LIN {X -403.787,Y 333.050,Z -17.519,A 0.015,B -0.000,C 180.000} C_DIS
LIN {X -401.252,Y 328.076,Z -17.721,A 0.015,B -0.000,C -180.000} C_DIS
LIN {X -395.738,Y 327.203,Z -17.924,A 0.015,B 0.000,C -180.000} C_DIS
LIN {X -391.790,Y 331.150,Z -18.126,A 0.015,B 0.000,C 180.000} C_DIS
LIN {X -392.664,Y 336.664,Z -18.328,A 0.015,B -0.000,C -180.000} C_DIS
LIN {X -397.638,Y 339.199,Z -18.531,A 0.015,B 0.000,C 180.000} C_DIS
LIN {X -398.507,Y 339.199,Z -18.561,A 0.015,B -0.000,C 180.000} C_DIS
LIN {X -399.336,Y 339.133,Z -18.590,A 0.015,B -0.000,C -180.000} C_DIS
LIN {X -399.692,Y 339.076,Z -18.603,A 0.015,B -0.000,C -180.000} C_DIS
LIN {X -400.552,Y 338.848,Z -18.634,A 0.015,B 0.000,C 180.000} C_DIS
LIN {X -400.596,Y 338.832,Z -18.635,A 0.015,B 0.000,C -180.000} C_DIS
LIN {X -401.281,Y 338.494,Z -18.662,A 0.015,B 0.000,C 180.000} C_DIS
LIN {X -401.404,Y 338.418,Z -18.667,A 0.015,B 0.000,C 180.000} C_DIS
LIN {X -402.842,Y 337.053,Z -18.737,A 0.015,B -0.000,C 180.000} C_DIS
LIN {X -402.866,Y 337.018,Z -18.738,A 0.015,B 0.000,C -180.000} C_DIS
LIN {X -403.753,Y 334.430,Z -18.835,A 0.015,B -0.000,C -180.000} C_DIS
LIN {X -403.779,Y 333.946,Z -18.852,A 0.015,B -0.000,C -180.000} C_DIS
LIN {X -403.787,Y 333.653,Z -18.862,A 0.015,B -0.000,C -180.000} C_DIS
LIN {X -403.787,Y 333.050,Z -18.883,A 0.015,B 0.000,C -180.000} C_DIS
LIN {X -401.252,Y 328.076,Z -19.086,A 0.015,B -0.000,C 180.000} C_DIS
LIN {X -395.738,Y 327.203,Z -19.288,A 0.015,B 0.000,C -180.000} C_DIS
LIN {X -391.790,Y 331.150,Z -19.491,A 0.015,B 0.000,C 180.000} C_DIS
LIN {X -392.664,Y 336.664,Z -19.693,A 0.015,B -0.000,C -180.000} C_DIS
LIN {X -397.638,Y 339.199,Z -19.895,A 0.015,B 0.000,C 180.000} C_DIS
LIN {X -398.507,Y 339.199,Z -19.926,A 0.015,B 0.000,C -180.000} C_DIS
LIN {X -399.336,Y 339.133,Z -19.955,A 0.015,B -0.000,C 180.000} C_DIS
LIN {X -399.692,Y 339.076,Z -19.967,A 0.015,B -0.000,C 180.000} C_DIS
LIN {X -400.552,Y 338.848,Z -19.998,A 0.015,B -0.000,C 180.000} C_DIS
LIN {X -400.596,Y 338.832,Z -20.000,A 0.015,B 0.000,C 180.000} C_DIS
LIN {X -400.134,Y 339.006,Z -20.000,A 0.015,B -0.000,C 180.000} C_DIS
LIN {X -398.924,Y 339.199,Z -20.000,A 0.015,B 0.000,C 180.000} C_DIS
LIN {X -213.196,Y 339.203,Z -20.000,A 0.015,B 0.000,C 180.000} C_DIS
LIN {X -213.589,Y 339.144,Z -20.000,A 0.015,B -0.000,C 180.000} C_DIS
LIN {X -214.096,Y 339.026,Z -20.000,A 0.015,B 0.000,C 180.000} C_DIS
LIN {X -215.185,Y 338.684,Z -20.000,A 0.015,B 0.000,C 180.000} C_DIS
LIN {X -215.676,Y 338.486,Z -20.000,A 0.015,B -0.000,C -180.000} C_DIS
LIN {X -226.923,Y 332.891,Z -20.000,A 0.015,B 0.000,C 180.000} C_DIS
LIN {X -227.590,Y 332.454,Z -20.000,A 0.015,B 0.000,C -180.000} C_DIS
LIN {X -228.678,Y 331.541,Z -20.000,A 0.015,B 0.000,C 180.000} C_DIS
LIN {X -228.854,Y 331.383,Z -20.000,A 0.015,B -0.000,C 180.000} C_DIS
LIN {X -237.260,Y 323.263,Z -20.000,A 0.015,B 0.000,C -180.000} C_DIS
LIN {X -237.740,Y 322.682,Z -20.000,A 0.015,B 0.000,C -180.000} C_DIS
LIN {X -238.689,Y 321.231,Z -20.000,A 0.015,B -0.000,C -180.000} C_DIS
LIN {X -238.828,Y 321.000,Z -20.000,A 0.015,B 0.000,C -180.000} C_DIS
LIN {X -243.976,Y 311.569,Z -20.000,A 0.015,B -0.000,C 180.000} C_DIS
LIN {X -244.137,Y 311.231,Z -20.000,A 0.015,B 0.000,C -180.000} C_DIS
LIN {X -244.732,Y 309.780,Z -20.000,A 0.015,B -0.000,C 180.000} C_DIS
LIN {X -244.946,Y 309.009,Z -20.000,A 0.015,B 0.000,C 180.000} C_DIS
LIN {X -246.389,Y 299.577,Z -20.000,A 0.015,B 0.000,C 180.000} C_DIS
LIN {X -246.415,Y 299.356,Z -20.000,A 0.015,B -0.000,C 180.000} C_DIS
LIN {X -246.509,Y 298.268,Z -20.000,A 0.015,B -0.000,C -180.000} C_DIS
CIRC {X -246.514,Y 297.749,Z -20.000,A 0.015,B 0.000,C -180.000},{X -246.439,Y 297.235,Z -20.000,A 0.015,B 0.000,C -180.000} C_DIS
LIN {X -245.041,Y 291.021,Z -20.000,A 0.015,B 0.000,C 180.000} C_DIS
LIN {X -245.028,Y 290.962,Z -20.000,A 0.015,B 0.000,C 180.000} C_DIS
LIN {X -244.067,Y 287.020,Z -20.000,A 0.015,B 0.000,C 180.000} C_DIS
LIN {X -243.752,Y 286.205,Z -20.000,A 0.015,B 0.000,C -180.000} C_DIS
LIN {X -242.372,Y 283.666,Z -20.000,A 0.015,B 0.000,C 180.000} C_DIS
LIN {X -242.162,Y 283.330,Z -20.000,A 0.015,B -0.000,C -180.000} C_DIS
LIN {X -239.169,Y 279.093,Z -20.000,A 0.015,B 0.000,C -180.000} C_DIS
LIN {X -239.003,Y 278.877,Z -20.000,A 0.015,B 0.000,C -180.000} C_DIS
LIN {X -237.090,Y 276.585,Z -20.000,A 0.015,B -0.000,C -180.000} C_DIS
LIN {X -236.752,Y 276.235,Z -20.000,A 0.015,B 0.000,C -180.000} C_DIS
LIN {X -236.388,Y 275.908,Z -20.000,A 0.015,B -0.000,C -180.000} C_DIS
LIN {X -236.084,Y 275.665,Z -20.000,A 0.015,B 0.000,C 180.000} C_DIS
LIN {X -232.452,Y 273.091,Z -20.000,A 0.015,B 0.000,C -180.000} C_DIS
LIN {X -232.331,Y 273.008,Z -20.000,A 0.015,B -0.000,C -180.000} C_DIS
LIN {X -229.064,Y 270.900,Z -20.000,A 0.015,B 0.000,C -180.000} C_DIS
LIN {X -228.750,Y 270.720,Z -20.000,A 0.015,B -0.000,C 180.000} C_DIS
LIN {X -227.172,Y 269.926,Z -20.000,A 0.015,B 0.000,C -180.000} C_DIS
LIN {X -226.775,Y 269.757,Z -20.000,A 0.015,B 0.000,C -180.000} C_DIS
LIN {X -224.725,Y 269.036,Z -20.000,A 0.015,B 0.000,C 180.000} C_DIS
LIN {X -224.251,Y 268.907,Z -20.000,A 0.015,B 0.000,C 180.000} C_DIS
LIN {X -219.172,Y 267.914,Z -20.000,A 0.015,B 0.000,C -180.000} C_DIS
LIN {X -218.973,Y 267.881,Z -20.000,A 0.015,B 0.000,C 180.000} C_DIS
LIN {X -215.345,Y 267.394,Z -20.000,A 0.015,B 0.000,C 180.000} C_DIS
LIN {X -214.895,Y 267.364,Z -20.000,A 0.015,B 0.000,C 180.000} C_DIS
LIN {X -178.617,Y 267.364,Z -20.000,A 0.015,B 0.000,C 180.000} C_DIS
LIN {X -178.167,Y 267.394,Z -20.000,A 0.015,B -0.000,C 180.000} C_DIS
LIN {X -174.539,Y 267.881,Z -20.000,A 0.015,B -0.000,C 180.000} C_DIS
LIN {X -174.340,Y 267.914,Z -20.000,A 0.015,B 0.000,C -180.000} C_DIS
LIN {X -169.261,Y 268.907,Z -20.000,A 0.015,B 0.000,C 180.000} C_DIS
LIN {X -168.860,Y 269.012,Z -20.000,A 0.015,B 0.000,C 180.000} C_DIS
LIN {X -167.472,Y 269.465,Z -20.000,A 0.015,B 0.000,C -180.000} C_DIS
LIN {X -167.129,Y 269.598,Z -20.000,A 0.015,B 0.000,C -180.000} C_DIS
LIN {X -165.283,Y 270.432,Z -20.000,A 0.015,B 0.000,C -180.000} C_DIS
LIN {X -164.859,Y 270.662,Z -20.000,A 0.015,B 0.000,C -180.000} C_DIS
LIN {X -161.562,Y 272.763,Z -20.000,A 0.015,B 0.000,C -180.000} C_DIS
LIN {X -161.461,Y 272.830,Z -20.000,A 0.015,B 0.000,C -180.000} C_DIS
LIN {X -158.559,Y 274.828,Z -20.000,A 0.015,B 0.000,C 180.000} C_DIS
LIN {X -158.397,Y 274.947,Z -20.000,A 0.015,B 0.000,C -180.000} C_DIS
LIN {X -156.938,Y 276.085,Z -20.000,A 0.015,B 0.000,C -180.000} C_DIS
LIN {X -156.452,Y 276.549,Z -20.000,A 0.015,B 0.000,C -180.000} C_DIS
LIN {X -155.008,Y 278.233,Z -20.000,A 0.015,B -0.000,C 180.000} C_DIS
LIN {X -154.823,Y 278.469,Z -20.000,A 0.015,B -0.000,C 180.000} C_DIS
LIN {X -151.360,Y 283.315,Z -20.000,A 0.015,B -0.000,C 180.000} C_DIS
LIN {X -151.140,Y 283.666,Z -20.000,A 0.015,B 0.000,C 180.000} C_DIS
LIN {X -149.760,Y 286.205,Z -20.000,A 0.015,B -0.000,C 180.000} C_DIS
LIN {X -149.440,Y 287.040,Z -20.000,A 0.015,B 0.000,C -180.000} C_DIS
LIN {X -147.117,Y 296.834,Z -20.000,A 0.015,B 0.000,C -180.000} C_DIS
LIN {X -147.030,Y 297.450,Z -20.000,A 0.015,B -0.000,C 180.000} C_DIS
LIN {X -146.995,Y 298.175,Z -20.000,A 0.015,B 0.000,C 180.000} C_DIS
LIN {X -147.027,Y 298.837,Z -20.000,A 0.015,B 0.000,C 180.000} C_DIS
LIN {X -148.481,Y 308.631,Z -20.000,A 0.015,B 0.000,C 180.000} C_DIS
LIN {X -148.624,Y 309.222,Z -20.000,A 0.015,B 0.000,C 180.000} C_DIS
LIN {X -149.116,Y 310.673,Z -20.000,A 0.015,B 0.000,C 180.000} C_DIS
LIN {X -149.349,Y 311.203,Z -20.000,A 0.015,B -0.000,C -180.000} C_DIS
LIN {X -154.682,Y 320.997,Z -20.000,A 0.015,B 0.000,C -180.000} C_DIS
LIN {X -154.822,Y 321.231,Z -20.000,A 0.015,B 0.000,C -180.000} C_DIS
LIN {X -155.772,Y 322.682,Z -20.000,A 0.015,B 0.000,C 180.000} C_DIS
LIN {X -156.247,Y 323.258,Z -20.000,A 0.015,B 0.000,C 180.000} C_DIS
LIN {X -163.722,Y 330.512,Z -20.000,A 0.015,B 0.000,C 180.000} C_DIS
LIN {X -163.842,Y 330.624,Z -20.000,A 0.015,B 0.000,C 180.000} C_DIS
LIN {X -165.860,Y 332.401,Z -20.000,A 0.015,B 0.000,C -180.000} C_DIS
LIN {X -166.589,Y 332.891,Z -20.000,A 0.015,B -0.000,C 180.000} C_DIS
LIN {X -177.836,Y 338.486,Z -20.000,A 0.015,B 0.000,C 180.000} C_DIS
LIN {X -178.194,Y 338.639,Z -20.000,A 0.015,B 0.000,C -180.000} C_DIS
LIN {X -178.919,Y 338.901,Z -20.000,A 0.015,B 0.000,C -180.000} C_DIS
LIN {X -179.549,Y 339.062,Z -20.000,A 0.015,B 0.000,C 180.000} C_DIS
LIN {X -180.468,Y 339.204,Z -20.000,A 0.015,B 0.000,C -180.000} C_DIS
LIN {X 4.865,Y 339.209,Z -20.000,A 0.015,B -0.000,C -180.000} C_DIS
LIN {X 5.937,Y 339.152,Z -20.000,A 0.015,B -0.000,C 180.000} C_DIS
LIN {X 6.802,Y 338.955,Z -20.000,A 0.015,B 0.000,C 180.000} C_DIS
LIN {X 7.069,Y 338.840,Z -20.000,A 0.015,B 0.000,C 180.000} C_DIS
LIN {X 7.374,Y 338.634,Z -20.000,A 0.015,B -0.000,C 180.000} C_DIS
LIN {X 9.664,Y 336.377,Z -20.000,A 0.015,B 0.000,C -180.000} C_DIS
LIN {X 9.898,Y 336.018,Z -20.000,A 0.015,B 0.000,C -180.000} C_DIS
LIN {X 10.072,Y 335.556,Z -20.000,A 0.015,B -0.000,C -180.000} C_DIS
LIN {X 10.265,Y 334.347,Z -20.000,A 0.015,B -0.000,C 180.000} C_DIS
LIN {X 10.273,Y 31.658,Z -20.000,A 0.015,B 0.000,C -180.000} C_DIS
LIN {X 8.905,Y 37.176,Z -20.000,A 0.015,B 0.000,C 180.000} C_DIS
LIN {X 8.665,Y 37.838,Z -20.000,A 0.015,B 0.000,C 180.000} C_DIS
LIN {X 7.997,Y 39.214,Z -20.000,A 0.015,B -0.000,C -180.000} C_DIS
LIN {X 7.843,Y 39.497,Z -20.000,A 0.015,B -0.000,C -180.000} C_DIS
LIN {X 2.038,Y 49.028,Z -20.000,A 0.015,B 0.000,C -180.000} C_DIS
LIN {X 1.811,Y 49.356,Z -20.000,A 0.015,B 0.000,C -180.000} C_DIS
LIN {X 0.937,Y 50.469,Z -20.000,A 0.015,B -0.000,C -180.000} C_DIS
LIN {X 0.391,Y 51.021,Z -20.000,A 0.015,B 0.000,C -180.000} C_DIS
LIN {X -7.442,Y 57.299,Z -20.000,A 0.015,B 0.000,C -180.000} C_DIS
LIN {X -7.813,Y 57.558,Z -20.000,A 0.015,B 0.000,C 180.000} C_DIS
LIN {X -8.481,Y 57.960,Z -20.000,A 0.015,B 0.000,C 180.000} C_DIS
LIN {X -9.249,Y 58.300,Z -20.000,A 0.015,B 0.000,C 180.000} C_DIS
LIN {X -19.102,Y 61.270,Z -20.000,A 0.015,B 0.000,C -180.000} C_DIS
LIN {X -19.977,Y 61.413,Z -20.000,A 0.015,B 0.000,C -180.000} C_DIS
LIN {X -22.516,Y 61.489,Z -20.000,A 0.015,B 0.000,C 180.000} C_DIS
LIN {X -22.912,Y 61.478,Z -20.000,A 0.015,B 0.000,C 180.000} C_DIS
LIN {X -28.717,Y 60.970,Z -20.000,A 0.015,B -0.000,C 180.000} C_DIS
LIN {X -29.063,Y 60.922,Z -20.000,A 0.015,B -0.000,C -180.000} C_DIS
LIN {X -31.966,Y 60.361,Z -20.000,A 0.015,B 0.000,C -180.000} C_DIS
LIN {X -32.711,Y 60.125,Z -20.000,A 0.015,B 0.000,C 180.000} C_DIS
LIN {X -36.585,Y 58.384,Z -20.000,A 0.015,B 0.000,C 180.000} C_DIS
LIN {X -36.742,Y 58.308,Z -20.000,A 0.015,B -0.000,C 180.000} C_DIS
LIN {X -40.593,Y 56.333,Z -20.000,A 0.015,B 0.000,C 180.000} C_DIS
LIN {X -40.908,Y 56.149,Z -20.000,A 0.015,B 0.000,C -180.000} C_DIS
LIN {X -42.316,Y 55.223,Z -20.000,A 0.015,B 0.000,C 180.000} C_DIS
LIN {X -42.641,Y 54.980,Z -20.000,A 0.015,B 0.000,C -180.000} C_DIS
LIN {X -44.193,Y 53.668,Z -20.000,A 0.015,B -0.000,C 180.000} C_DIS
LIN {X -44.555,Y 53.312,Z -20.000,A 0.015,B 0.000,C -180.000} C_DIS
LIN {X -48.485,Y 48.820,Z -20.000,A 0.015,B 0.000,C -180.000} C_DIS
LIN {X -48.631,Y 48.641,Z -20.000,A 0.015,B -0.000,C 180.000} C_DIS
LIN {X -50.408,Y 46.306,Z -20.000,A 0.015,B 0.000,C 180.000} C_DIS
LIN {X -50.645,Y 45.950,Z -20.000,A 0.015,B 0.000,C 180.000} C_DIS
LIN {X -68.791,Y 14.550,Z -20.000,A 0.015,B 0.000,C 180.000} C_DIS
LIN {X -68.995,Y 14.133,Z -20.000,A 0.015,B 0.000,C -180.000} C_DIS
LIN {X -70.620,Y 10.143,Z -20.000,A 0.015,B 0.000,C -180.000} C_DIS
LIN {X -70.685,Y 9.967,Z -20.000,A 0.015,B 0.000,C -180.000} C_DIS
LIN {X -72.182,Y 5.614,Z -20.000,A 0.015,B 0.000,C 180.000} C_DIS
LIN {X -72.291,Y 5.221,Z -20.000,A 0.015,B -0.000,C -180.000} C_DIS
LIN {X -72.602,Y 3.770,Z -20.000,A 0.015,B 0.000,C -180.000} C_DIS
LIN {X -72.660,Y 3.396,Z -20.000,A 0.015,B -0.000,C -180.000} C_DIS
LIN {X -72.875,Y 1.219,Z -20.000,A 0.015,B 0.000,C 180.000} C_DIS
LIN {X -72.886,Y 0.696,Z -20.000,A 0.015,B 0.000,C -180.000} C_DIS
LIN {X -72.517,Y -5.833,Z -20.000,A 0.015,B 0.000,C -180.000} C_DIS
LIN {X -72.500,Y -6.030,Z -20.000,A 0.015,B 0.000,C -180.000} C_DIS
LIN {X -72.249,Y -8.206,Z -20.000,A 0.015,B 0.000,C -180.000} C_DIS
LIN {X -72.158,Y -8.686,Z -20.000,A 0.015,B 0.000,C 180.000} C_DIS
LIN {X -71.966,Y -9.411,Z -20.000,A 0.015,B 0.000,C 180.000} C_DIS
LIN {X -71.856,Y -9.753,Z -20.000,A 0.015,B 0.000,C 180.000} C_DIS
LIN {X -70.762,Y -12.612,Z -20.000,A 0.015,B 0.000,C 180.000} C_DIS
LIN {X -70.674,Y -12.821,Z -20.000,A 0.015,B 0.000,C 180.000} C_DIS
LIN {X -68.645,Y -17.217,Z -20.000,A 0.015,B 0.000,C 180.000} C_DIS
LIN {X -68.494,Y -17.507,Z -20.000,A 0.015,B 0.000,C -180.000} C_DIS
LIN {X -67.645,Y -18.958,Z -20.000,A 0.015,B 0.000,C -180.000} C_DIS
LIN {X -67.514,Y -19.164,Z -20.000,A 0.015,B 0.000,C -180.000} C_DIS
LIN {X -66.750,Y -20.278,Z -20.000,A 0.015,B 0.000,C -180.000} C_DIS
LIN {X -66.282,Y -20.825,Z -20.000,A 0.015,B 0.000,C 180.000} C_DIS
LIN {X -59.766,Y -26.970,Z -20.000,A 0.015,B 0.000,C -180.000} C_DIS
LIN {X -59.608,Y -27.111,Z -20.000,A 0.015,B 0.000,C -180.000} C_DIS
LIN {X -58.519,Y -28.016,Z -20.000,A 0.015,B 0.000,C 180.000} C_DIS
CIRC {X -58.085,Y -28.322,Z -20.000,A 0.015,B 0.000,C -180.000},{X -57.609,Y -28.557,Z -20.000,A 0.015,B -0.000,C 180.000} C_DIS
LIN {X -50.808,Y -31.266,Z -20.000,A 0.015,B 0.000,C 180.000} C_DIS
LIN {X -342.732,Y -31.266,Z -20.000,A 0.015,B 0.000,C -180.000} C_DIS
LIN {X -336.289,Y -28.753,Z -20.000,A 0.015,B 0.000,C -180.000} C_DIS
LIN {X -335.783,Y -28.505,Z -20.000,A 0.015,B 0.000,C -180.000} C_DIS
LIN {X -335.057,Y -28.072,Z -20.000,A 0.015,B -0.000,C 180.000} C_DIS
LIN {X -334.481,Y -27.638,Z -20.000,A 0.015,B 0.000,C 180.000} C_DIS
LIN {X -329.122,Y -22.621,Z -20.000,A 0.015,B 0.000,C 180.000} C_DIS
LIN {X -329.059,Y -22.561,Z -20.000,A 0.015,B -0.000,C 180.000} C_DIS
LIN {X -326.883,Y -20.415,Z -20.000,A 0.015,B 0.000,C 180.000} C_DIS
LIN {X -326.355,Y -19.743,Z -20.000,A 0.015,B 0.000,C 180.000} C_DIS
LIN {X -325.035,Y -17.535,Z -20.000,A 0.015,B 0.000,C 180.000} C_DIS
LIN {X -324.867,Y -17.215,Z -20.000,A 0.015,B 0.000,C 180.000} C_DIS
LIN {X -322.511,Y -12.105,Z -20.000,A 0.015,B 0.000,C 180.000} C_DIS
LIN {X -322.392,Y -11.812,Z -20.000,A 0.015,B 0.000,C -180.000} C_DIS
LIN {X -321.509,Y -9.305,Z -20.000,A 0.015,B 0.000,C -180.000} C_DIS
LIN {X -321.344,Y -8.614,Z -20.000,A 0.015,B 0.000,C -180.000} C_DIS
LIN {X -321.018,Y -6.074,Z -20.000,A 0.015,B 0.000,C -180.000} C_DIS
LIN {X -320.995,Y -5.833,Z -20.000,A 0.015,B 0.000,C 180.000} C_DIS
LIN {X -320.626,Y 0.696,Z -20.000,A 0.015,B 0.000,C -180.000} C_DIS
LIN {X -320.630,Y 1.140,Z -20.000,A 0.015,B -0.000,C 180.000} C_DIS
LIN {X -320.739,Y 2.591,Z -20.000,A 0.015,B -0.000,C 180.000} C_DIS
LIN {X -320.790,Y 2.973,Z -20.000,A 0.015,B -0.000,C 180.000} C_DIS
LIN {X -321.206,Y 5.149,Z -20.000,A 0.015,B -0.000,C 180.000} C_DIS
LIN {X -321.329,Y 5.614,Z -20.000,A 0.015,B -0.000,C -180.000} C_DIS
LIN {X -322.710,Y 9.630,Z -20.000,A 0.015,B 0.000,C -180.000} C_DIS
LIN {X -322.763,Y 9.773,Z -20.000,A 0.015,B -0.000,C -180.000} C_DIS
LIN {X -324.328,Y 13.737,Z -20.000,A 0.015,B 0.000,C 180.000} C_DIS
LIN {X -324.544,Y 14.184,Z -20.000,A 0.015,B -0.000,C 180.000} C_DIS
LIN {X -342.684,Y 45.663,Z -20.000,A 0.015,B 0.000,C -180.000} C_DIS
LIN {X -342.906,Y 46.000,Z -20.000,A 0.015,B 0.000,C -180.000} C_DIS
LIN {X -344.864,Y 48.619,Z -20.000,A 0.015,B -0.000,C -180.000} C_DIS
LIN {X -345.015,Y 48.806,Z -20.000,A 0.015,B 0.000,C -180.000} C_DIS
LIN {X -348.417,Y 52.738,Z -20.000,A 0.015,B 0.000,C -180.000} C_DIS
LIN {X -348.646,Y 52.978,Z -20.000,A 0.015,B 0.000,C 180.000} C_DIS
LIN {X -350.214,Y 54.466,Z -20.000,A 0.015,B 0.000,C -180.000} C_DIS
LIN {X -350.587,Y 54.773,Z -20.000,A 0.015,B 0.000,C 180.000} C_DIS
LIN {X -352.038,Y 55.801,Z -20.000,A 0.015,B -0.000,C -180.000} C_DIS
LIN {X -352.424,Y 56.037,Z -20.000,A 0.015,B -0.000,C -180.000} C_DIS
LIN {X -356.264,Y 58.049,Z -20.000,A 0.015,B 0.000,C 180.000} C_DIS
LIN {X -356.429,Y 58.130,Z -20.000,A 0.015,B 0.000,C -180.000} C_DIS
LIN {X -360.783,Y 60.117,Z -20.000,A 0.015,B -0.000,C 180.000} C_DIS
LIN {X -361.546,Y 60.361,Z -20.000,A 0.015,B -0.000,C -180.000} C_DIS
LIN {X -364.449,Y 60.922,Z -20.000,A 0.015,B 0.000,C 180.000} C_DIS
LIN {X -364.780,Y 60.969,Z -20.000,A 0.015,B 0.000,C -180.000} C_DIS
LIN {X -370.222,Y 61.469,Z -20.000,A 0.015,B 0.000,C 180.000} C_DIS
LIN {X -370.612,Y 61.483,Z -20.000,A 0.015,B -0.000,C 180.000} C_DIS
LIN {X -373.514,Y 61.413,Z -20.000,A 0.015,B 0.000,C -180.000} C_DIS
LIN {X -374.398,Y 61.274,Z -20.000,A 0.015,B 0.000,C 180.000} C_DIS
LIN {X -383.583,Y 58.541,Z -20.000,A 0.015,B 0.000,C -180.000} C_DIS
LIN {X -383.906,Y 58.427,Z -20.000,A 0.015,B -0.000,C 180.000} C_DIS
LIN {X -384.908,Y 58.014,Z -20.000,A 0.015,B -0.000,C 180.000} C_DIS
LIN {X -385.728,Y 57.532,Z -20.000,A 0.015,B -0.000,C -180.000} C_DIS
LIN {X -393.895,Y 51.027,Z -20.000,A 0.015,B 0.000,C -180.000} C_DIS
LIN {X -394.449,Y 50.469,Z -20.000,A 0.015,B 0.000,C -180.000} C_DIS
LIN {X -395.323,Y 49.356,Z -20.000,A 0.015,B 0.000,C -180.000} C_DIS
LIN {X -395.550,Y 49.028,Z -20.000,A 0.015,B 0.000,C -180.000} C_DIS
LIN {X -401.355,Y 39.497,Z -20.000,A 0.015,B -0.000,C -180.000} C_DIS
LIN {X -401.509,Y 39.214,Z -20.000,A 0.015,B 0.000,C -180.000} C_DIS
LIN {X -402.177,Y 37.838,Z -20.000,A 0.015,B 0.000,C 180.000} C_DIS
LIN {X -402.417,Y 37.176,Z -20.000,A 0.015,B 0.000,C -180.000} C_DIS
LIN {X -403.779,Y 31.685,Z -20.000,A 0.015,B -0.000,C -180.000} C_DIS
LIN {X -403.787,Y 333.800,Z -20.000,A 0.015,B -0.000,C -180.000} C_DIS
LIN {X -403.730,Y 334.871,Z -20.000,A 0.015,B 0.000,C -180.000} C_DIS
LIN {X -403.533,Y 335.736,Z -20.000,A 0.015,B -0.000,C 180.000} C_DIS
LIN {X -403.418,Y 336.003,Z -20.000,A 0.015,B -0.000,C 180.000} C_DIS
LIN {X -403.034,Y 336.500,Z -19.830,A 0.015,B 0.000,C 180.000} C_DIS
LIN {X -402.624,Y 336.714,Z -19.365,A 0.015,B 0.000,C 180.000} C_DIS
LIN {X -402.458,Y 336.753,Z -18.730,A 0.015,B 0.000,C -180.000} C_DIS
$VEL.CP = 1.00000
LIN {X -402.458,Y 336.753,Z 11.000,A 0.015,B 0.000,C 180.000} C_DIS
$VEL.CP = 1.00000
LIN {X -212.830,Y 109.416,Z 11.000,A 0.015,B 0.000,C 180.000} C_DIS
$VEL.CP = 0.10000
LIN {X -212.830,Y 109.416,Z -8.231,A 0.015,B 0.000,C -180.000} C_DIS
LIN {X -212.668,Y 109.398,Z -8.853,A 0.015,B -0.000,C 180.000} C_DIS
LIN {X -212.222,Y 109.369,Z -9.316,A 0.015,B 0.000,C 180.000} C_DIS
LIN {X -211.606,Y 109.385,Z -9.500,A 0.015,B 0.000,C -180.000} C_DIS
LIN {X -206.370,Y 113.409,Z -9.744,A 0.015,B -0.000,C 180.000} C_DIS
LIN {X -207.958,Y 119.819,Z -9.988,A 0.015,B 0.000,C -180.000} C_DIS
LIN {X -214.468,Y 120.933,Z -10.232,A 0.015,B 0.000,C 180.000} C_DIS
LIN {X -218.097,Y 115.415,Z -10.476,A 0.015,B -0.000,C -180.000} C_DIS
LIN {X -214.495,Y 109.879,Z -10.720,A 0.015,B 0.000,C -180.000} C_DIS
LIN {X -207.980,Y 110.960,Z -10.964,A 0.015,B 0.000,C 180.000} C_DIS
LIN {X -206.360,Y 117.363,Z -11.208,A 0.015,B -0.000,C 180.000} C_DIS
LIN {X -211.577,Y 121.413,Z -11.452,A 0.015,B 0.000,C 180.000} C_DIS
LIN {X -217.378,Y 118.256,Z -11.696,A 0.015,B 0.000,C -180.000} C_DIS
LIN {X -216.810,Y 111.676,Z -11.940,A 0.015,B 0.000,C -180.000} C_DIS
LIN {X -210.554,Y 109.559,Z -12.185,A 0.015,B 0.000,C -180.000} C_DIS
LIN {X -206.108,Y 114.443,Z -12.429,A 0.015,B 0.000,C 180.000} C_DIS
LIN {X -208.801,Y 120.473,Z -12.673,A 0.015,B 0.000,C 180.000} C_DIS
LIN {X -215.405,Y 120.423,Z -12.917,A 0.015,B 0.000,C 180.000} C_DIS
LIN {X -218.005,Y 114.352,Z -13.161,A 0.015,B -0.000,C 180.000} C_DIS
LIN {X -213.485,Y 109.537,Z -13.405,A 0.015,B 0.000,C 180.000} C_DIS
LIN {X -207.262,Y 111.749,Z -13.649,A 0.015,B 0.000,C -180.000} C_DIS
LIN {X -206.795,Y 118.337,Z -13.893,A 0.015,B -0.000,C 180.000} C_DIS
LIN {X -212.643,Y 121.404,Z -14.137,A 0.015,B 0.000,C 180.000} C_DIS
LIN {X -217.798,Y 117.275,Z -14.381,A 0.015,B 0.000,C 180.000} C_DIS
LIN {X -216.080,Y 110.898,Z -14.625,A 0.015,B 0.000,C -180.000} C_DIS
LIN {X -209.549,Y 109.917,Z -14.869,A 0.015,B -0.000,C 180.000} C_DIS
LIN {X -206.033,Y 115.507,Z -15.113,A 0.015,B 0.000,C 180.000} C_DIS
LIN {X -209.745,Y 120.969,Z -15.357,A 0.015,B 0.000,C 180.000} C_DIS
LIN {X -216.237,Y 119.756,Z -15.601,A 0.015,B 0.000,C -180.000} C_DIS
LIN {X -217.728,Y 113.322,Z -15.845,A 0.015,B -0.000,C 180.000} C_DIS
LIN {X -212.430,Y 109.378,Z -16.089,A 0.015,B 0.000,C -180.000} C_DIS
LIN {X -206.694,Y 112.652,Z -16.333,A 0.015,B 0.000,C 180.000} C_DIS
LIN {X -207.395,Y 119.219,Z -16.577,A 0.015,B 0.000,C -180.000} C_DIS
LIN {X -213.692,Y 121.208,Z -16.821,A 0.015,B 0.000,C -180.000} C_DIS
LIN {X -218.038,Y 116.236,Z -17.065,A 0.015,B 0.000,C 180.000} C_DIS
LIN {X -215.224,Y 110.261,Z -17.310,A 0.015,B 0.000,C -180.000} C_DIS
LIN {X -208.623,Y 110.445,Z -17.554,A 0.015,B -0.000,C -180.000} C_DIS
LIN {X -206.146,Y 116.568,Z -17.798,A 0.015,B 0.000,C -180.000} C_DIS
LIN {X -210.762,Y 121.290,Z -18.042,A 0.015,B 0.000,C 180.000} C_DIS
LIN {X -216.939,Y 118.953,Z -18.286,A 0.015,B -0.000,C 180.000} C_DIS
LIN {X -217.273,Y 112.357,Z -18.530,A 0.015,B 0.000,C -180.000} C_DIS
LIN {X -211.364,Y 109.408,Z -18.774,A 0.015,B 0.000,C 180.000} C_DIS
LIN {X -206.294,Y 113.641,Z -19.018,A 0.015,B 0.000,C -180.000} C_DIS
LIN {X -208.140,Y 119.982,Z -19.262,A 0.015,B 0.000,C -180.000} C_DIS
LIN {X -214.690,Y 120.831,Z -19.506,A 0.015,B 0.000,C -180.000} C_DIS
LIN {X -218.092,Y 115.171,Z -19.750,A 0.015,B 0.000,C 180.000} C_DIS
LIN {X -214.270,Y 109.785,Z -19.994,A 0.015,B 0.000,C 180.000} C_DIS
LIN {X -207.804,Y 111.129,Z -20.238,A 0.015,B -0.000,C -180.000} C_DIS
LIN {X -206.444,Y 117.592,Z -20.482,A 0.015,B -0.000,C 180.000} C_DIS
LIN {X -211.820,Y 121.427,Z -20.726,A 0.015,B 0.000,C -180.000} C_DIS
LIN {X -217.489,Y 118.039,Z -20.970,A 0.015,B -0.000,C -180.000} C_DIS
LIN {X -216.656,Y 111.487,Z -21.214,A 0.015,B 0.000,C -180.000} C_DIS
LIN {X -210.319,Y 109.625,Z -21.458,A 0.015,B 0.000,C -180.000} C_DIS
LIN {X -206.074,Y 114.684,Z -21.702,A 0.015,B 0.000,C 180.000} C_DIS
LIN {X -209.009,Y 120.601,Z -21.946,A 0.015,B -0.000,C -180.000} C_DIS
LIN {X -215.605,Y 120.284,Z -22.190,A 0.015,B 0.000,C 180.000} C_DIS
LIN {X -217.958,Y 114.113,Z -22.435,A 0.015,B 0.000,C -180.000} C_DIS
LIN {X -213.247,Y 109.484,Z -22.679,A 0.015,B 0.000,C -180.000} C_DIS
LIN {X -207.118,Y 111.946,Z -22.923,A 0.015,B 0.000,C 180.000} C_DIS
LIN {X -206.918,Y 118.547,Z -23.167,A 0.015,B -0.000,C 180.000} C_DIS
LIN {X -212.886,Y 121.376,Z -23.411,A 0.015,B -0.000,C 180.000} C_DIS
LIN {X -217.869,Y 117.042,Z -23.655,A 0.015,B -0.000,C -180.000} C_DIS
LIN {X -215.895,Y 110.740,Z -23.899,A 0.015,B 0.000,C 180.000} C_DIS
LIN {X -209.329,Y 110.023,Z -24.143,A 0.015,B 0.000,C -180.000} C_DIS
LIN {X -206.042,Y 115.751,Z -24.387,A 0.015,B -0.000,C 180.000} C_DIS
LIN {X -209.972,Y 121.058,Z -24.631,A 0.015,B 0.000,C 180.000} C_DIS
LIN {X -216.410,Y 119.584,Z -24.875,A 0.015,B 0.000,C 180.000} C_DIS
LIN {X -217.639,Y 113.095,Z -25.119,A 0.015,B 0.000,C 180.000} C_DIS
LIN {X -212.186,Y 109.368,Z -25.363,A 0.015,B 0.000,C 180.000} C_DIS
LIN {X -206.587,Y 112.871,Z -25.607,A 0.015,B 0.000,C -180.000} C_DIS
LIN {X -207.553,Y 119.404,Z -25.851,A 0.015,B 0.000,C -180.000} C_DIS
LIN {X -213.926,Y 121.138,Z -26.095,A 0.015,B 0.000,C 180.000} C_DIS
LIN {X -218.067,Y 115.994,Z -26.339,A 0.015,B 0.000,C -180.000} C_DIS
LIN {X -215.014,Y 110.138,Z -26.583,A 0.015,B 0.000,C -180.000} C_DIS
LIN {X -208.425,Y 110.588,Z -26.827,A 0.015,B 0.000,C 180.000} C_DIS
LIN {X -206.198,Y 116.806,Z -27.071,A 0.015,B 0.000,C -180.000} C_DIS
LIN {X -211.002,Y 121.338,Z -27.315,A 0.015,B 0.000,C -180.000} C_DIS
LIN {X -217.079,Y 118.753,Z -27.560,A 0.015,B 0.000,C 180.000} C_DIS
LIN {X -217.146,Y 112.149,Z -27.804,A 0.015,B 0.000,C 180.000} C_DIS
LIN {X -211.122,Y 109.441,Z -28.048,A 0.015,B 0.000,C 180.000} C_DIS
LIN {X -206.227,Y 113.875,Z -28.292,A 0.015,B -0.000,C -180.000} C_DIS
LIN {X -208.329,Y 120.136,Z -28.536,A 0.015,B 0.000,C -180.000} C_DIS
LIN {X -214.907,Y 120.720,Z -28.780,A 0.015,B -0.000,C 180.000} C_DIS
LIN {X -218.078,Y 114.927,Z -29.024,A 0.015,B 0.000,C 180.000} C_DIS
LIN {X -214.041,Y 109.700,Z -29.268,A 0.015,B 0.000,C 180.000} C_DIS
LIN {X -207.635,Y 111.305,Z -29.512,A 0.015,B 0.000,C 180.000} C_DIS
LIN {X -206.537,Y 117.817,Z -29.756,A 0.015,B 0.000,C -180.000} C_DIS
LIN {X -212.064,Y 121.432,Z -30.000,A 0.015,B 0.000,C -180.000} C_DIS
LIN {X -214.073,Y 121.432,Z -30.000,A 0.015,B 0.000,C -180.000} C_DIS
CIRC {X -215.997,Y 120.322,Z -30.000,A 0.015,B 0.000,C -180.000},{X -215.999,Y 118.101,Z -30.000,A 0.015,B -0.000,C 180.000} C_DIS
LIN {X -214.838,Y 116.087,Z -30.000,A 0.015,B 0.000,C 180.000} C_DIS
CIRC {X -213.799,Y 115.047,Z -30.000,A 0.015,B 0.000,C 180.000},{X -212.379,Y 114.666,Z -30.000,A 0.015,B 0.000,C 180.000} C_DIS
LIN {X -181.119,Y 114.666,Z -30.000,A 0.015,B -0.000,C 180.000} C_DIS
CIRC {X -179.701,Y 115.046,Z -30.000,A 0.015,B 0.000,C 180.000},{X -178.662,Y 116.084,Z -30.000,A 0.015,B 0.000,C 180.000} C_DIS
LIN {X -177.499,Y 118.096,Z -30.000,A 0.015,B 0.000,C -180.000} C_DIS
CIRC {X -177.498,Y 120.320,Z -30.000,A 0.015,B 0.000,C -180.000},{X -179.424,Y 121.432,Z -30.000,A 0.015,B 0.000,C 180.000} C_DIS
LIN {X -212.064,Y 121.432,Z -30.000,A 0.015,B 0.000,C -180.000} C_DIS
CIRC {X -215.508,Y 122.484,Z -30.000,A 0.015,B -0.000,C -180.000},{X -217.776,Y 125.281,Z -30.000,A 0.015,B 0.000,C -180.000} C_DIS
CIRC {X -219.946,Y 128.117,Z -30.000,A 0.015,B 0.000,C -180.000},{X -223.260,Y 129.446,Z -30.000,A 0.015,B 0.000,C -180.000} C_DIS
CIRC {X -226.456,Y 129.803,Z -30.000,A 0.015,B 0.000,C -180.000},{X -229.654,Y 130.146,Z -30.000,A 0.015,B 0.000,C -180.000} C_DIS
CIRC {X -231.451,Y 129.229,Z -30.000,A 0.015,B 0.000,C -180.000},{X -231.344,Y 127.213,Z -30.000,A 0.015,B 0.000,C 180.000} C_DIS
CIRC {X -228.587,Y 123.273,Z -30.000,A 0.015,B -0.000,C 180.000},{X -225.983,Y 119.230,Z -30.000,A 0.015,B 0.000,C 180.000} C_DIS
CIRC {X -223.488,Y 115.120,Z -30.000,A 0.015,B -0.000,C -180.000},{X -221.056,Y 110.972,Z -30.000,A 0.015,B 0.000,C -180.000} C_DIS
CIRC {X -217.951,Y 107.863,Z -30.000,A 0.015,B 0.000,C 180.000},{X -213.707,Y 106.725,Z -30.000,A 0.015,B -0.000,C -180.000} C_DIS
LIN {X -179.805,Y 106.725,Z -30.000,A 0.015,B 0.000,C -180.000} C_DIS
CIRC {X -175.556,Y 107.863,Z -30.000,A 0.015,B 0.000,C 180.000},{X -172.444,Y 110.973,Z -30.000,A 0.015,B 0.000,C -180.000} C_DIS
CIRC {X -170.014,Y 115.114,Z -30.000,A 0.015,B 0.000,C -180.000},{X -167.530,Y 119.222,Z -30.000,A 0.015,B -0.000,C 180.000} C_DIS
CIRC {X -164.940,Y 123.265,Z -30.000,A 0.015,B -0.000,C -180.000},{X -162.197,Y 127.207,Z -30.000,A 0.015,B -0.000,C 180.000} C_DIS
CIRC {X -162.093,Y 129.225,Z -30.000,A 0.015,B 0.000,C -180.000},{X -163.893,Y 130.142,Z -30.000,A 0.015,B 0.000,C 180.000} C_DIS
CIRC {X -167.567,Y 129.748,Z -30.000,A 0.015,B 0.000,C 180.000},{X -171.239,Y 129.335,Z -30.000,A 0.015,B -0.000,C 180.000} C_DIS
CIRC {X -174.922,Y 129.018,Z -30.000,A 0.015,B -0.000,C -180.000},{X -178.617,Y 128.912,Z -30.000,A 0.015,B -0.000,C 180.000} C_DIS
LIN {X -214.895,Y 128.911,Z -30.000,A 0.015,B -0.000,C 180.000} C_DIS
CIRC {X -218.599,Y 129.018,Z -30.000,A 0.015,B -0.000,C 180.000},{X -222.291,Y 129.336,Z -30.000,A 0.015,B -0.000,C 180.000} C_DIS
LIN {X -223.260,Y 129.446,Z -30.000,A 0.015,B 0.000,C -180.000} C_DIS
CIRC {X -226.330,Y 130.760,Z -30.000,A 0.015,B -0.000,C -180.000},{X -228.172,Y 133.545,Z -30.000,A 0.015,B 0.000,C 180.000} C_DIS
CIRC {X -229.976,Y 136.341,Z -30.000,A 0.015,B 0.000,C 180.000},{X -232.988,Y 137.754,Z -30.000,A 0.015,B 0.000,C 180.000} C_DIS
CIRC {X -240.220,Y 138.961,Z -30.000,A 0.015,B -0.000,C 180.000},{X -247.436,Y 140.259,Z -30.000,A 0.015,B 0.000,C -180.000} C_DIS
CIRC {X -249.157,Y 139.464,Z -30.000,A 0.015,B 0.000,C 180.000},{X -248.977,Y 137.577,Z -30.000,A 0.015,B 0.000,C -180.000} C_DIS
CIRC {X -246.164,Y 134.353,Z -30.000,A 0.015,B 0.000,C -180.000},{X -243.314,Y 131.161,Z -30.000,A 0.015,B 0.000,C 180.000} C_DIS
CIRC {X -240.519,Y 127.919,Z -30.000,A 0.015,B -0.000,C -180.000},{X -237.877,Y 124.552,Z -30.000,A 0.015,B 0.000,C 180.000} C_DIS
CIRC {X -234.395,Y 119.527,Z -30.000,A 0.015,B 0.000,C -180.000},{X -231.284,Y 114.264,Z -30.000,A 0.015,B 0.000,C -180.000} C_DIS
CIRC {X -228.333,Y 108.914,Z -30.000,A 0.015,B 0.000,C 180.000},{X -225.316,Y 103.601,Z -30.000,A 0.015,B -0.000,C 180.000} C_DIS
CIRC {X -222.211,Y 100.492,Z -30.000,A 0.015,B 0.000,C -180.000},{X -217.967,Y 99.354,Z -30.000,A 0.015,B 0.000,C -180.000} C_DIS
LIN {X -175.551,Y 99.354,Z -30.000,A 0.015,B 0.000,C 180.000} C_DIS

; Continue running program as cascaded execution
Machining1()

END
